FUNCTION_BLOCK TaitBryanAngleOrientation EXTENDS AngleSequenceOrientation
VAR_INPUT
END_VAR
VAR_OUTPUT
END_VAR
VAR
	Angles_ : ARRAY [0..2] OF LREAL;
	Sequence_ : TaitBryanAngleSequence;
END_VAR

METHOD PUBLIC  GetAngle : LREAL
VAR_INPUT
	I : UINT;
END_VAR
VAR
	Dim : Dimension;
END_VAR
IF I >= Length THEN
	GetAngle := 0;
	RETURN;
END_IF

Dim := GetDimension(I);

IF Dim >= Length THEN
	GetAngle := 0;
	RETURN;
END_IF

GetAngle := Angles_[Dim];
END_METHOD

METHOD PUBLIC GetDimension : Dimension
VAR_INPUT
	I : UINT;
END_VAR
VAR
	Dims : ARRAY [0..2] OF Dimension;
END_VAR
IF I >= Length THEN
	GetDimension := 0;
	RETURN;
END_IF

Dims := GetDimensions();
GetDimension := Dims[I];
END_METHOD

METHOD PUBLIC GetDimensions : ARRAY [0..2] OF Dimension
VAR_INPUT
END_VAR
CASE Sequence OF
	TaitBryanAngleSequence.XYZ:
		GetDimensions[0] := 0;
		GetDimensions[1] := 1;
		GetDimensions[2] := 2;
	TaitBryanAngleSequence.XZY:
		GetDimensions[0] := 0;
		GetDimensions[1] := 2;
		GetDimensions[2] := 1;
	TaitBryanAngleSequence.YXZ:
		GetDimensions[0] := 1;
		GetDimensions[1] := 0;
		GetDimensions[2] := 2;
	TaitBryanAngleSequence.YZX:
		GetDimensions[0] := 1;
		GetDimensions[1] := 2;
		GetDimensions[2] := 0;
	TaitBryanAngleSequence.ZXY:
		GetDimensions[0] := 2;
		GetDimensions[1] := 0;
		GetDimensions[2] := 1;
	TaitBryanAngleSequence.ZYX:
		GetDimensions[0] := 2;
		GetDimensions[1] := 1;
		GetDimensions[2] := 0;
	ELSE
		GetDimensions[0] := 0;
		GetDimensions[1] := 0;
		GetDimensions[2] := 0;
END_CASE
END_METHOD

PROPERTY Length : UINT
GET
Length := 3;
END_GET
END_PROPERTY

PROPERTY PUBLIC RxDeg : LREAL
GET
RxDeg := 180 * Angles_[0] / PI;
END_GET
SET
Angles_[0] := PI * RxDeg / 180;
END_SET
END_PROPERTY

PROPERTY PUBLIC RxRad : LREAL
GET
RxRad := Angles_[0];
END_GET
SET
Angles_[0] := RxRad;
END_SET
END_PROPERTY

PROPERTY PUBLIC RyDeg : LREAL
GET
RyDeg := 180 * Angles_[1] / PI;
END_GET
SET
Angles_[1] := PI * RyDeg / 180;
END_SET
END_PROPERTY

PROPERTY PUBLIC RyRad : LREAL
GET
RyRad := Angles_[1];
END_GET
SET
Angles_[1] := RyRad;
END_SET
END_PROPERTY

PROPERTY PUBLIC RzDeg : LREAL
GET
RzDeg := 180 * Angles_[2] / PI;
END_GET
SET
Angles_[2] := PI * RzDeg / 180;
END_SET
END_PROPERTY

PROPERTY PUBLIC RzRad : LREAL
GET
RzRad := Angles_[2];
END_GET
SET
Angles_[2] := RzRad;
END_SET
END_PROPERTY

PROPERTY PUBLIC Sequence : TaitBryanAngleSequence
GET
Sequence := Sequence_;
END_GET
SET
Sequence_ := Sequence;
END_SET
END_PROPERTY

METHOD PUBLIC SetAngle : BOOL
VAR_INPUT
	I : UINT;
	Val : LREAL;
END_VAR
VAR
	Dim : Dimension;
END_VAR
IF I >= Length THEN
	SetAngle := FALSE;
	RETURN;
END_IF

Dim := GetDimension(I);

IF Dim >= Length THEN
	SetAngle := FALSE;
	RETURN;
END_IF

SetAngle := TRUE;

Angles_[Dim] := Val;
END_METHOD

METHOD PUBLIC SetFromComponentsDeg
VAR_INPUT
	Rx : LREAL;
	Ry : LREAL;
	Rz : LREAL;
	Seq : TaitBryanAngleSequence;
END_VAR
RxDeg := Rx;
RyDeg := Ry;
RzDeg := Rz;
Sequence := Seq;
END_METHOD

METHOD PUBLIC SetFromComponentsRad
VAR_INPUT
	Rx : LREAL;
	Ry : LREAL;
	Rz : LREAL;
	Seq : TaitBryanAngleSequence;
END_VAR
RxRad := Rx;
RyRad := Ry;
RzRad := Rz;
Sequence := Seq;
END_METHOD

END_FUNCTION_BLOCK

(* stored: Version 1.1.0.1, ProductVersion 3.1.4024.9
   POU TaitBryanAngleOrientation: Id {30f16bb7-b6a8-07ba-01fe-7fa9cf8edcd3}, SpecialFunc None
   Folder Getters: Id {d092d2bb-44ff-015b-23d0-0cd0696517ea}
   Folder Properties: Id {cfe678ce-52d8-0d59-378d-9d7a9f94d78e}
   Folder Setters: Id {476f1314-1760-0491-162a-ca22b126dafb}
   Method GetAngle: Id {f6726e47-c5fb-0990-0956-4dd56856561f}
   Method GetDimension: Id {69e98eb8-908f-0785-2692-8746de432a97}
   Method GetDimensions: Id {2cd7e7e1-f488-048d-091d-9e023d75faaa}
   Property Length: Id {a6ac7c86-1428-0662-043d-544990228d08}
   Get Get: Id {2a85c423-ef9b-08d9-2079-0739d9af36a0}
   Property RxDeg: Id {202974e2-8c00-0fea-3ea3-e7c0eef9724c}
   Get Get: Id {b77c4288-df7d-087d-1a88-477a2518b241}
   Set Set: Id {88eafb0b-2c6d-0979-33df-28e4a08cccd2}
   Property RxRad: Id {8c7a8fb7-996d-0655-0d2c-d6e6dfff0ccb}
   Get Get: Id {55821b3b-df54-0b0e-3aec-5a2afcde2db5}
   Set Set: Id {d0bb744d-82a1-0de4-12bc-802f8660aaac}
   Property RyDeg: Id {71278da6-8344-0821-398c-4a19e65bf722}
   Get Get: Id {d8139ec5-0086-0127-0a6c-e1ab20004c64}
   Set Set: Id {521419e4-aeb9-0e67-3406-cc3086e090a7}
   Property RyRad: Id {de7cefc7-a31a-0dea-206f-3553e6978e35}
   Get Get: Id {84c391e8-c14c-0f77-0a7c-dbe8ae38b1b7}
   Set Set: Id {9f9b4df5-6f3a-019b-0abc-2692dd5a467a}
   Property RzDeg: Id {d87122d9-49a2-0517-18b6-eefd59b51d18}
   Get Get: Id {807a4354-cd23-0b9b-0128-62683afc992e}
   Set Set: Id {e7f1f502-f4e7-0ddc-347f-d814a3c9f4f3}
   Property RzRad: Id {8e1cae5d-0f96-0804-190f-1b7cddb4c154}
   Get Get: Id {8c7eaa5a-ecd8-0ed8-0647-52e2c1bc6519}
   Set Set: Id {a08a6319-ebd0-0b30-3846-60b7569e33c0}
   Property Sequence: Id {bdbbf1cc-9abf-0851-1958-c67ed62108f2}
   Get Get: Id {c01ca441-f7fa-0521-25d3-1e68afd2ff61}
   Set Set: Id {fd12c575-2803-0ce1-33b8-c23c25cde2d3}
   Method SetAngle: Id {4ebf317e-4620-0dbb-0fd2-2805540c84d9}
   Method SetFromComponentsDeg: Id {426c64c2-25ed-0ee8-1928-5154abb51fe0}
   Method SetFromComponentsRad: Id {73c29634-84a1-0471-382d-dc6b1c8f59e3} *)
